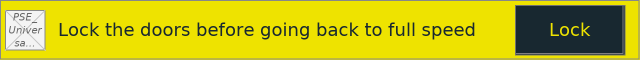
VISUALIZATION AOIHeaderKeySwitchFrame  // 640x60
VAR_IN_OUT
	btnDoorsLock : BOOL;
END_VAR
    Label (55,10 440x40), "Lock the doors before going back to full speed"
    Button (515,5 110x50), "Lock"
        toggle btnDoorsLock
    Image (5,10 40x40), image: PSE_UniversalBlocks.IP_EventSeverity.error
END_VISUALIZATION

(* stored: Version 1.1.0.1, ProductVersion 3.1.4024.9
   Visu AOIHeaderKeySwitchFrame: Id {198e8440-0b28-464b-a79a-ea52aca712cf} *)
